FUNCTION_BLOCK ARRAY2VALUES_8_INT (* Service Interface Function Block Type *)
  (* Description: Copyright (c) 2014 Profactor GmbH, HR Agrartechnik GmbH This program and the accompanying materials are made available under the terms of the Eclipse Public License 2.0 which is available at https://www.eclipse.org/legal/epl-2.0/ SPDX-License-Identifier: EPL-2.0 *)
  (* Version 1.0, 2026-03-30, Franz Höpfinger, HR Agrartechnik GmbH, copy ARRAY2VALUES_2_LREAL and made this block *)
  PACKAGE eclipse4diac::convert;
  {SET_ATTRIBUTE(eclipse4diac::core::GenericClassName, 'GEN_ARRAY2VALUES')}
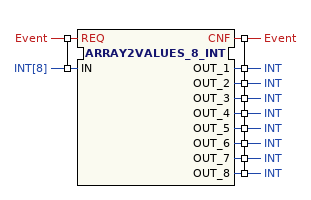
  EVENT_INPUT
    REQ WITH IN; (* Service Request *)
  END_EVENT
  EVENT_OUTPUT
    CNF WITH OUT_1, OUT_2, OUT_3, OUT_4, OUT_5, OUT_6, OUT_7, OUT_8; (* Confirmation of Requested Service *)
  END_EVENT
  VAR_INPUT
    IN : ARRAY [0..7] OF INT; (* Array input *)
  END_VAR
  VAR_OUTPUT
    OUT_1 : INT; (* output number 1 *)
    OUT_2 : INT; (* output number 2 *)
    OUT_3 : INT; (* output number 3 *)
    OUT_4 : INT; (* output number 4 *)
    OUT_5 : INT; (* output number 5 *)
    OUT_6 : INT; (* output number 6 *)
    OUT_7 : INT; (* output number 7 *)
    OUT_8 : INT; (* output number 8 *)
  END_VAR
END_FUNCTION_BLOCK
